{attribute 'qualified_only'}
VAR_GLOBAL

IX_START AT %I*: BOOL;
IX_STOP AT %I*:	BOOL;
	
END_VAR

(* stored: Version 1.1.0.1, ProductVersion 3.1.4024.6
   GVL StartStop: Id {37cb43e4-e979-4317-8127-9cb6a323c694} *)
